Omron CX-Programmer project 新工程 (CX-Programmer 9.42)

# PLC 新PLC1: CP1H XA

## Global symbols (name address type ; comment)
0.00 BOOL  ; 启动/急停开关
0.01 BOOL  ; 光电开关
0.02 BOOL  ; 强制上升开关
0.03 BOOL  ; 强制下降开关
0.04 BOOL  ; 强制上升开关
0.05 BOOL  ; 强制下降开关
0.06 BOOL  ; 强制下降开关
10.00 BOOL  ; 卷帘门上升
10.01 BOOL  ; 卷帘门下降
10.02 BOOL  ; 报警
16.00 BOOL  ; 中间继电器1
17.00 BOOL  ; 中间继电器2
18.00 BOOL  ; 上行程开关
19.00 BOOL  ; 下行程开关
200.00 BOOL  ; 报警中继
C0001 BOOL  ; 计数器
T0000 BOOL  ; 延时3s
T0002 BOOL  ; 延时10s下降
T0003 BOOL  ; 延时判断是否有车
T0004 BOOL  ; 上升时间
T0005 BOOL  ; 下降时间
T0006 BOOL  ; 15s
T0007 BOOL  ; 报警闪烁

## Program 新程序1 (cyclic task 0)

### Section 段1

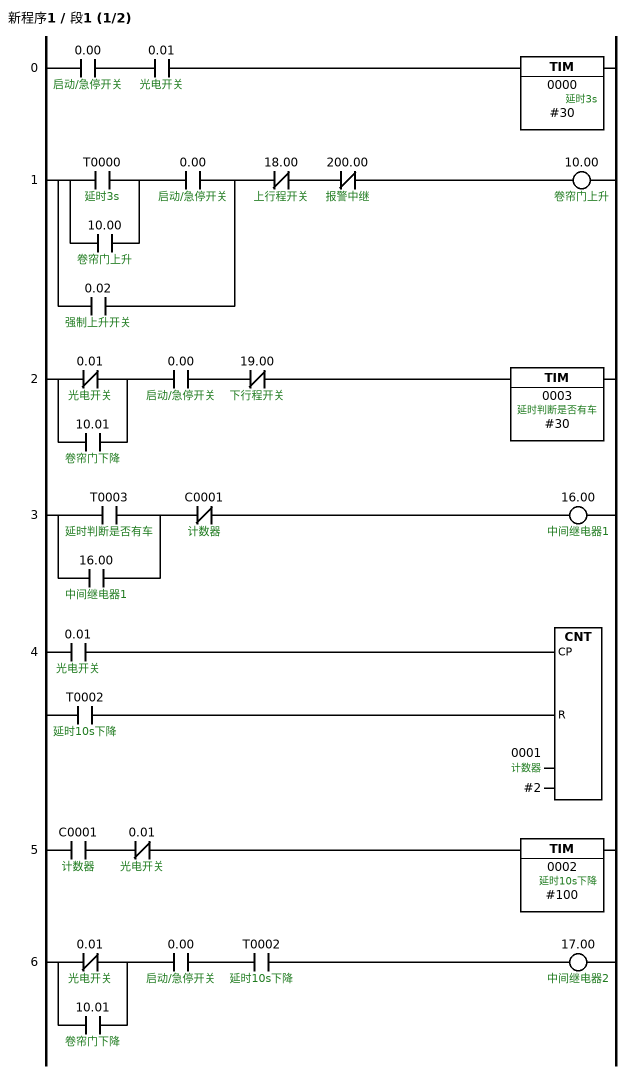
; rung 0
LD 0.00  ; 启动/急停开关
AND 0.01  ; 光电开关
TIM 0000 #30  ; 延时3s
; rung 1
LD T0000  ; 延时3s
OR 10.00  ; 卷帘门上升
AND 0.00  ; 启动/急停开关
OR 0.02  ; 强制上升开关
ANDNOT 18.00  ; 上行程开关
ANDNOT 200.00  ; 报警中继
OUT 10.00  ; 卷帘门上升
; rung 2
LDNOT 0.01  ; 光电开关
OR 10.01  ; 卷帘门下降
AND 0.00  ; 启动/急停开关
ANDNOT 19.00  ; 下行程开关
TIM 0003 #30  ; 延时判断是否有车
; rung 3
LD T0003  ; 延时判断是否有车
OR 16.00  ; 中间继电器1
ANDNOT C0001  ; 计数器
OUT 16.00  ; 中间继电器1
; rung 4
LD 0.01  ; 光电开关
LD T0002  ; 延时10s下降
CNT 0001 #2  ; 计数器
; rung 5
LD C0001  ; 计数器
ANDNOT 0.01  ; 光电开关
TIM 0002 #100  ; 延时10s下降
; rung 6
LDNOT 0.01  ; 光电开关
OR 10.01  ; 卷帘门下降
AND 0.00  ; 启动/急停开关
AND T0002  ; 延时10s下降
OUT 17.00  ; 中间继电器2

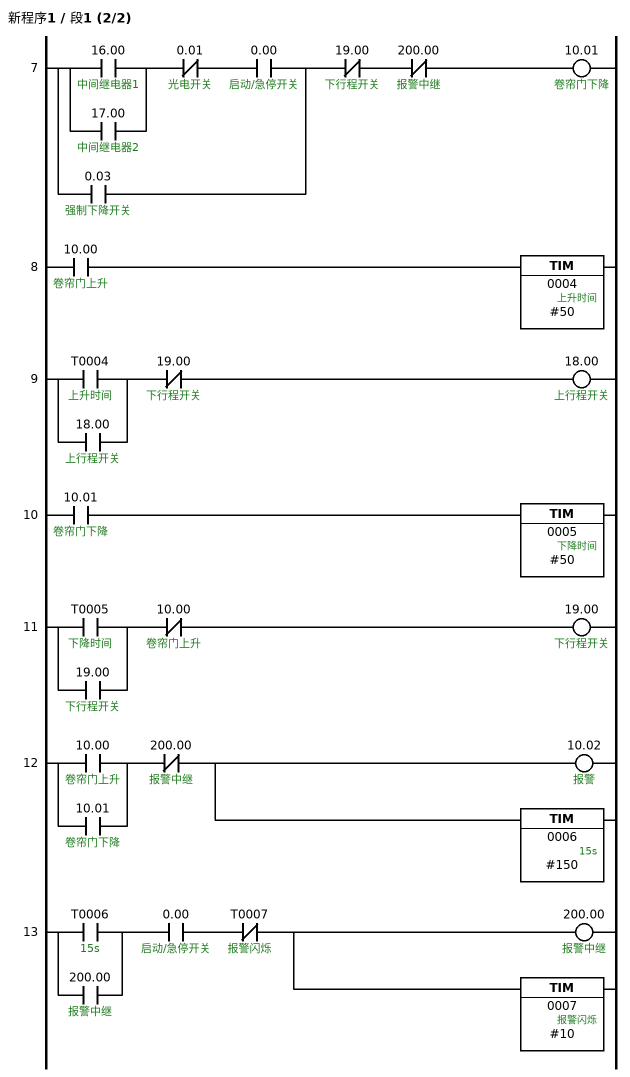
; rung 7
LD 16.00  ; 中间继电器1
OR 17.00  ; 中间继电器2
ANDNOT 0.01  ; 光电开关
AND 0.00  ; 启动/急停开关
OR 0.03  ; 强制下降开关
ANDNOT 19.00  ; 下行程开关
ANDNOT 200.00  ; 报警中继
OUT 10.01  ; 卷帘门下降
; rung 8
LD 10.00  ; 卷帘门上升
TIM 0004 #50  ; 上升时间
; rung 9
LD T0004  ; 上升时间
OR 18.00  ; 上行程开关
ANDNOT 19.00  ; 下行程开关
OUT 18.00  ; 上行程开关
; rung 10
LD 10.01  ; 卷帘门下降
TIM 0005 #50  ; 下降时间
; rung 11
LD T0005  ; 下降时间
OR 19.00  ; 下行程开关
ANDNOT 10.00  ; 卷帘门上升
OUT 19.00  ; 下行程开关
; rung 12
LD 10.00  ; 卷帘门上升
OR 10.01  ; 卷帘门下降
ANDNOT 200.00  ; 报警中继
OUT 10.02  ; 报警
TIM 0006 #150  ; 15s
; rung 13
LD T0006  ; 15s
OR 200.00  ; 报警中继
AND 0.00  ; 启动/急停开关
ANDNOT T0007  ; 报警闪烁
OUT 200.00  ; 报警中继
TIM 0007 #10  ; 报警闪烁

### Section END
; rung 0
END(001)